TYPE E_CodeType :
(
	E_NONE,
	E_PACK,
	E_INTERIM,
	E_OUTER,
	E_CASE

);
END_TYPE

(* stored: Version 1.1.0.1
   DUT E_CodeType: Id {c110f819-a9fb-41b3-bd8b-89eb095e6f4f} *)
